// TIA Portal V20 export
TYPE "LCFL_typeMaintenance"
TITLE = HMI data for LCFL_Maintenance / HMI-Daten für LCFL_Maintenance
// Data type for HMI data / HMI-Daten für LCFL_Maintenance
   STRUCT
      operatingTimeAct : Real;   // Tatsächliche Betriebszeit des Antriebs [h] / Actual operating time of the drive [h]
      operatingTimeLimit : Real;   // Max. Grenze der Betriebszeit [h] / Max. limit of the operating time [h]
      operatingTimeReached { ExternalWritable := 'False'} : Bool;   // 1: Die tatsächlichen Betriebsstunden haben ihre Grenze erreicht oder überschritten (wenn Grenzwert > 0) / 1: The actual operating hours have reached or exceeded their limit (if limit > 0)
      cycleTimeAct : Real;   // Tatsächliche Zykluszeit des Antriebs [h] / Actual cycle time of the drive [h]
      cycleTimeLimit : Real;   // Max. Grenze der Zykluszeit [h] / Max. limit of the cycle time [h]
      cycleTimeReached { ExternalWritable := 'False'} : Bool;   // 1: Die tatsächliche Zykluszeit hat ihre Grenze erreicht oder überschritten (wenn Grenzwert > 0) / 1: The actual cycle time have reached or exceeded their limit (if limit > 0)
      switchCounterAct : UDInt;   // Tatsächliche Anzahl der Schaltungen des Antriebs / Actual number of switches of the drive
      switchCounterLimit : UDInt;   // Max. Grenzwert des Schalterzählers / Max. limit of switch counter
      switchCounterReached { ExternalWritable := 'False'} : Bool;   // 1: Die tatsächliche Anzahl der Zustandswechsel hat seine Grenze erreicht oder überschritten (wenn Grenzwert > 0) / 1: The actual switch counter has reached or exceeded its limit (if limit > 0)
      alarmCounterAct : UDInt;   // Tatsächliche Anzahl der Alarmmeldungen des Antriebs / Actual number of alarms of the drive
      alarmCounterLimit : UDInt;   // Max. Grenzwert des Alarmzählers / Max. limit of alarm counter
      alarmCounterReached { ExternalWritable := 'False'} : Bool;   // 1: Der aktuelle Alarmzähler hat seinen Grenzwert erreicht oder überschritten (wenn Grenzwert > 0) / 1: The actual alarm counter has reached or exceeded its limit (if limit > 0)
   END_STRUCT;
END_TYPE
